// TIA Portal V20 export
FUNCTION "Vis_Button_wide外观变量映射" : Void   // FC5, LAD
{ S7_Optimized_Access := 'TRUE' }
// stored: SetENOAutomatically false
   VAR_TEMP
      x1 : Bool;
   END_VAR
BEGIN

REGION Network 1
   // 轴1轴2点动速度映射
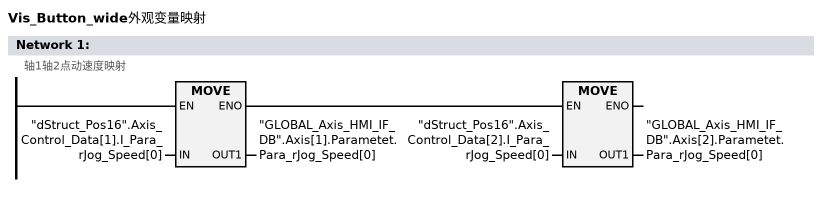
   RUNG wire#powerrail
      Move(in := "dStruct_Pos16".Axis_Control_Data[1].I_Para_rJog_Speed[0], out1 => "GLOBAL_Axis_HMI_IF_DB".Axis[1].Parametet.Para_rJog_Speed[0])
      Move(in := "dStruct_Pos16".Axis_Control_Data[2].I_Para_rJog_Speed[0], out1 => "GLOBAL_Axis_HMI_IF_DB".Axis[2].Parametet.Para_rJog_Speed[0])
   END_RUNG
   // the same network as SCL:
   "GLOBAL_Axis_HMI_IF_DB".Axis[1].Parametet.Para_rJog_Speed[0] := "dStruct_Pos16".Axis_Control_Data[1].I_Para_rJog_Speed[0];
   "GLOBAL_Axis_HMI_IF_DB".Axis[2].Parametet.Para_rJog_Speed[0] := "dStruct_Pos16".Axis_Control_Data[2].I_Para_rJog_Speed[0];
END_REGION

REGION Network 2 (SCL)
   "HMI变量汇总".Vis_Button_wideX1 := "IF_HMI_FB_IDB".IF.HMI[1].Vis_Button_wide.%X1;
   "HMI变量汇总".Vis_Button_wideX2 := "IF_HMI_FB_IDB".IF.HMI[1].Vis_Button_wide.%X2;
   "HMI变量汇总".Vis_Button_wideX3 := "IF_HMI_FB_IDB".IF.HMI[1].Vis_Button_wide.%X3;
   "HMI变量汇总".Vis_Button_wideX4 := "IF_HMI_FB_IDB".IF.HMI[1].Vis_Button_wide.%X4;
   "HMI变量汇总".Vis_Button_wideX5 := "IF_HMI_FB_IDB".IF.HMI[1].Vis_Button_wide.%X5;
   "HMI变量汇总".Vis_Button_wideX6 := "IF_HMI_FB_IDB".IF.HMI[1].Vis_Button_wide.%X6;
   "HMI变量汇总".Vis_Button_wideX7 := "IF_HMI_FB_IDB".IF.HMI[1].Vis_Button_wide.%X7;
   "HMI变量汇总".Vis_Button_wideX8 := "IF_HMI_FB_IDB".IF.HMI[1].Vis_Button_wide.%X8;
   "HMI变量汇总".Vis_Button_wideX9 := "IF_HMI_FB_IDB".IF.HMI[1].Vis_Button_wide.%X9;
   "HMI变量汇总".Vis_Button_wideX10 := "IF_HMI_FB_IDB".IF.HMI[1].Vis_Button_wide.%X10;
   "HMI变量汇总".Vis_Button_wideX11 := "IF_HMI_FB_IDB".IF.HMI[1].Vis_Button_wide.%X11;
   "HMI变量汇总".Vis_Button_wideX12 := "IF_HMI_FB_IDB".IF.HMI[1].Vis_Button_wide.%X12;

   "HMI变量汇总".Vis_Button_small1 := "IF_HMI_FB_IDB".IF.HMI[1].Vis_Button_small.%X1;
   "HMI变量汇总".Vis_Button_small2 := "IF_HMI_FB_IDB".IF.HMI[1].Vis_Button_small.%X2;
   "HMI变量汇总".Vis_Button_small3 := "IF_HMI_FB_IDB".IF.HMI[1].Vis_Button_small.%X3;
   "HMI变量汇总".Vis_Button_small4 := "IF_HMI_FB_IDB".IF.HMI[1].Vis_Button_small.%X4;
   "HMI变量汇总".Vis_Button_small5 := "IF_HMI_FB_IDB".IF.HMI[1].Vis_Button_small.%X5;
   "HMI变量汇总".Vis_Button_small6 := "IF_HMI_FB_IDB".IF.HMI[1].Vis_Button_small.%X6;
   "HMI变量汇总".Vis_Button_small7 := "IF_HMI_FB_IDB".IF.HMI[1].Vis_Button_small.%X7;
   "HMI变量汇总".Vis_Button_small8 := "IF_HMI_FB_IDB".IF.HMI[1].Vis_Button_small.%X8;
   "HMI变量汇总".Vis_Button_small9 := "IF_HMI_FB_IDB".IF.HMI[1].Vis_Button_small.%X9;
   "HMI变量汇总".Vis_Button_small10 := "IF_HMI_FB_IDB".IF.HMI[1].Vis_Button_small.%X10;
   "HMI变量汇总".Vis_Button_small11 := "IF_HMI_FB_IDB".IF.HMI[1].Vis_Button_small.%X11;
   "HMI变量汇总".Vis_Button_small12 := "IF_HMI_FB_IDB".IF.HMI[1].Vis_Button_small.%X12;




   #x1 := "IF_HMI_FB_IDB".IF.StateHeader_ForHMIAnimation[1].%X0;
   #x1 := "IF_HMI_FB_IDB".IF.StateHeader_ForHMIAnimation[1].%X1;
   #x1 := "IF_HMI_FB_IDB".IF.StateHeader_ForHMIAnimation[1].%X2;
   #x1 := "IF_HMI_FB_IDB".IF.StateHeader_ForHMIAnimation[1].%X3;
   #x1 := "IF_HMI_FB_IDB".IF.StateHeader_ForHMIAnimation[1].%X4;
   #x1 := "IF_HMI_FB_IDB".IF.StateHeader_ForHMIAnimation[1].%X5;
   #x1 := "IF_HMI_FB_IDB".IF.StateHeader_ForHMIAnimation[1].%X6;
   #x1 := "IF_HMI_FB_IDB".IF.StateHeader_ForHMIAnimation[1].%X7;
   #x1 := "IF_HMI_FB_IDB".IF.StateHeader_ForHMIAnimation[1].%X8;
   #x1 := "IF_HMI_FB_IDB".IF.StateHeader_ForHMIAnimation[1].%X9;
   #x1 := "IF_HMI_FB_IDB".IF.StateHeader_ForHMIAnimation[1].%X10;
   #x1 := "IF_HMI_FB_IDB".IF.StateHeader_ForHMIAnimation[1].%X11;
   #x1 := "IF_HMI_FB_IDB".IF.StateHeader_ForHMIAnimation[1].%X12;
   #x1 := "IF_HMI_FB_IDB".IF.StateHeader_ForHMIAnimation[1].%X13;
   #x1 := "IF_HMI_FB_IDB".IF.StateHeader_ForHMIAnimation[1].%X14;
   #x1 := "IF_HMI_FB_IDB".IF.StateHeader_ForHMIAnimation[1].%X15;
END_REGION
END_FUNCTION
